// TIA Portal V17 export
FUNCTION "FC_FanGasControl" : Void   // FC, LAD
{ S7_Optimized_Access := 'TRUE' }
BEGIN

REGION Network 1: 风机输出
   // 风机运行按常开+风机故障反馈常闭→风机运行线圈；手动选择MOVE自动输出或MUL手动频率×2→控制输出
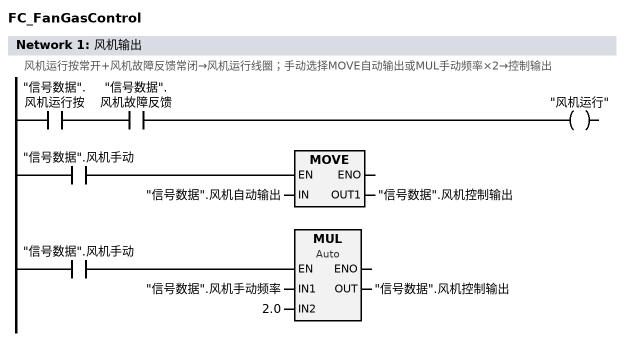
   RUNG wire#powerrail
      Contact( "信号数据".风机运行按 )
      Contact( "信号数据".风机故障反馈 )
      Coil( "风机运行" )
   END_RUNG
   RUNG wire#powerrail
      Contact( "信号数据".风机手动 )
      Move(in := "信号数据".风机自动输出, out1 => "信号数据".风机控制输出)
   END_RUNG
   RUNG wire#powerrail
      Contact( "信号数据".风机手动 )
      Mul(in1 := "信号数据".风机手动频率, in2 := 2.0, out => "信号数据".风机控制输出)
   END_RUNG
   // the same network as SCL:
   "风机运行" := "信号数据".风机运行按 AND "信号数据".风机故障反馈;
   IF "信号数据".风机手动 THEN
       "信号数据".风机控制输出 := "信号数据".风机自动输出;
       "信号数据".风机控制输出 := "信号数据".风机手动频率 * 2.0;
   END_IF;
END_REGION
END_FUNCTION
